// TwinCAT 3 PLC project SampleProject
// ProgramVersion: 3.1.4022.1
// libraries:
//   Tc2_Standard, * (Beckhoff Automation GmbH)
//   Tc2_System, * (Beckhoff Automation GmbH)
//   Tc2_Utilities, * (Beckhoff Automation GmbH)
//   Tc3_Module, * (Beckhoff Automation GmbH)
//   Tc3_PLCopen_OpcUa, * (Beckhoff Automation GmbH)
// project tree:
//   / PlcTask.TcTTO
//   POUs/ MAIN.TcPOU, PRG_HA_SingleNode.TcPOU
//   POUs/Multiple Nodes/ FB_HistoryUpdate_INT.TcPOU, FB_HistoryUpdate_LREAL.TcPOU, PRG_HA_MultipleNodes.TcPOU
// real-time tasks:
//   TASK PlcTask: cycle T#10ms, priority 20, ADS port 350

CONFIGURATION SampleProject
    RESOURCE PLC ON TwinCAT3
        TASK PlcTask(INTERVAL := T#10ms, PRIORITY := 20);
        PROGRAM MAIN WITH PlcTask : MAIN;
    END_RESOURCE
END_CONFIGURATION

// ---- POUs/MAIN.TcPOU
PROGRAM MAIN
VAR
	i : INT;
END_VAR

i := i + 1;

PRG_HA_SingleNode();	// call sample for UA_HistoryUpdate
PRG_HA_MultipleNodes();	// call sample for UA_HistoryUpdate with multiple nodes

END_PROGRAM

// ---- POUs/PRG_HA_SingleNode.TcPOU
//| use case:
//| One variable is specified for historical access. 
//| Its values of each task cycle should be updated to data storage.
PROGRAM PRG_HA_SingleNode
VAR CONSTANT
	// These connection and namespace settings need to be adapted to the runtime environment
	cOpcUaServerUrl		: STRING(MAX_STRING_LENGTH) := 'opc.tcp://localhost:4840';
	cNamespaceUri		: STRING(MAX_STRING_LENGTH) := 'urn:BeckhoffAutomation:Ua:PLC1';
	cBufferSize			: UINT := 1000;
END_VAR
VAR
	// Variable for HistorcalAccess
	{attribute 'OPC.UA.DA' := '1'}
	nMyValue : INT;	
	
	// state machine declarations 
	nState					: INT;
	bStart					: BOOL;			//Set True to start this sample.
	bSample					: BOOL := TRUE;	//Set True if data should be sampled.
	bStop					: BOOL;			//Set True to stop the sampling and close the connection afterwards.
	bError					: BOOL;
	nErrorID				: DWORD;
	
	// Declarations for UA_Connect
	fbUAConnect				: UA_Connect;
	stSessionConnectInfo 	: ST_UASessionConnectInfo;
	nConnectionHdl			: DWORD;
	
	// Declarations for UA_GetNamespaceIndex
	fbUAGetNamespaceIndex	: UA_GetNamespaceIndex;
	nNamespaceIndex			: UINT;
	
	// Declarations for UA_NodeGetHandle
	fbUANodeGetHandle		: UA_NodeGetHandle;
	sNodeIdentifier			: STRING(MAX_STRING_LENGTH) := 'PRG_HA_SingleNode.nMyValue'; // change to node identifier
	NodeID					: ST_UANodeID;
	nNodeHdl				: DWORD;
	
	// Declarations for UA_HistoryUpdate
	fbUAHistoryUpdate		: UA_HistoryUpdate;
	aDataValues				: ARRAY [1..cBufferSize] OF UAHADataValue(ValueSize:=SIZEOF(nMyValue));
	aValueErrorIDs			: ARRAY [1..cBufferSize] OF DWORD;
	nCounter				: UINT := 1;
	
	// Declarations for UA_NodeReleaseHandle
	fbUANodeReleaseHandle	: UA_NodeReleaseHandle;
	
	// Declarations for UA_Disconnect
	fbUADisconnect			: UA_Disconnect;
END_VAR

nMyValue := nMyValue + 1;

CASE nState OF
0:	//Idle
	IF bStart THEN  // the opc ua server need to be startet
		bStart				:= FALSE;
		bError				:= FALSE;
		nErrorID			:= 0;
		nCounter			:= 1;

		stSessionConnectInfo.tConnectTimeout 		:= T#1M;
		stSessionConnectInfo.tSessionTimeout 		:= T#1M;
		stSessionConnectInfo.sApplicationName		:= '';
		stSessionConnectInfo.eSecurityMode 			:= eUASecurityMsgMode_None;
		stSessionConnectInfo.eSecurityPolicyUri 	:= eUASecurityPolicy_None;
		stSessionConnectInfo.eTransportProfileUri	:= eUATransportProfileUri_UATcp;
		
		nState := 1;
	END_IF

1: //Open UA Session
	fbUAConnect(	Execute 			:= TRUE,
					ServerUrl			:= cOpcUaServerUrl,
					SessionConnectInfo	:= stSessionConnectInfo,
					Timeout				:= T#5S,
					ConnectionHdl 		=> nConnectionHdl );
		
	IF NOT fbUAConnect.Busy THEN
		IF NOT fbUAConnect.Error THEN
			nState 			:= 2;
		ELSE
			bError 			:= TRUE;
			nErrorID		:= fbUAConnect.ErrorID;
			nConnectionHdl 	:= 0;
			nState 			:= 0; //Idle
		END_IF
		fbUAConnect(Execute := FALSE);
	END_IF

2: //Get NS Index
	fbUAGetNamespaceIndex(	Execute 			:= TRUE,
							ConnectionHdl		:= nConnectionHdl,
							NamespaceUri		:= cNamespaceUri,
							NamespaceIndex		=> nNamespaceIndex );
		
	IF NOT fbUAGetNamespaceIndex.Busy THEN
		IF NOT fbUAGetNamespaceIndex.Error THEN
			nState 			:= 3;
		ELSE
			bError 			:= TRUE;
			nErrorID		:= fbUAGetNamespaceIndex.ErrorID;
			nState			:= 6; //Close Connection
		END_IF
		fbUAGetNamespaceIndex(Execute := FALSE);
	END_IF
	
3: //Get Node Handle
	NodeID.eIdentifierType 	:= eUAIdentifierType_String;
	NodeID.nNamespaceIndex 	:= nNamespaceIndex;
	NodeID.sIdentifier		:= sNodeIdentifier;
	
	fbUANodeGetHandle(	Execute 			:= TRUE,
						ConnectionHdl 		:= nConnectionHdl,
						NodeID 				:= NodeID,
						NodeHdl				=> nNodeHdl );
		
	IF NOT fbUANodeGetHandle.Busy THEN
		IF NOT fbUANodeGetHandle.Error THEN
			nState 			:= 4;
		ELSE
			bError  		:= TRUE;
			nErrorID 		:= fbUANodeGetHandle.ErrorID;
			nState 			:= 6; //Close Connection
		END_IF
		fbUANodeGetHandle(Execute := FALSE);
	END_IF
	
4: //UA_HistoryUpdate
	IF bSample THEN
		aDataValues[nCounter].Value				:= ADR(nMyValue);
		aDataValues[nCounter].StatusCode 		:= UAHAUpdateStatusCode.HistorianRaw;
		aDataValues[nCounter].ServerTimeStamp 	:= F_GetSystemTime();
		aDataValues[nCounter].SourceTimeStamp 	:= aDataValues[nCounter].ServerTimeStamp;	
		nCounter := nCounter + 1;
		
		IF nCounter > cBufferSize THEN
			fbUAHistoryUpdate.Execute := TRUE;
			nCounter := 1;
		END_IF
	END_IF
	
	fbUAHistoryUpdate(	Execute 			:= , //already set above
						ConnectionHdl 		:= nConnectionHdl,
						NodeHdl 			:= nNodeHdl,
						PerformInsert 		:= TRUE,
						PerformReplace 		:= FALSE,
						DataValueCount 		:= cBufferSize,
						DataValues	 		:= aDataValues,
						ValueErrorIDs 		:= aValueErrorIDs );
						
	IF NOT fbUAHistoryUpdate.Busy THEN
		IF NOT fbUAHistoryUpdate.Error THEN 
			IF bStop THEN
				bStop		:= FALSE;
				nState 		:= 5;
			END_IF
		ELSE
			bError 			:= TRUE;
			nErrorID 		:= fbUAHistoryUpdate.ErrorID;
			nState 			:= 5; //Release Node Handle
		END_IF
		fbUAHistoryUpdate(	Execute			:= FALSE, 			
							DataValues	 	:= aDataValues,
							ValueErrorIDs 	:= aValueErrorIDs);
	END_IF

5: //Release Node Handle
	fbUANodeReleaseHandle(	Execute 			:= TRUE,
							ConnectionHdl 		:= nConnectionHdl,
							NodeHdl 			:= nNodeHdl );
		
	IF NOT fbUANodeReleaseHandle.Busy THEN
		IF fbUANodeReleaseHandle.Error THEN
			bError 		:= TRUE;
			nErrorID 	:= fbUANodeReleaseHandle.ErrorID;
		END_IF
		fbUANodeReleaseHandle(Execute := FALSE);
		nState 			:= 6; //Close Connection
	END_IF

6: //Close Session
	fbUADisconnect( Execute := TRUE, ConnectionHdl := nConnectionHdl );
		
	IF NOT fbUADisconnect.Busy THEN
		IF fbUADisconnect.Error THEN
			bError 			:= TRUE;
			nErrorID 		:= fbUADisconnect.ErrorID;
			nConnectionHdl 	:= 0;
		END_IF
		fbUADisconnect(Execute := FALSE);
		nState := 0;
	END_IF
END_CASE

END_PROGRAM

// ---- POUs/Multiple Nodes/PRG_HA_MultipleNodes.TcPOU
//| use case:
//| Three variables are specified for historical access. 
//| Every three seconds their values should be updated to data storage for one second long.
PROGRAM PRG_HA_MultipleNodes
VAR CONSTANT
	// These connection and namespace settings need to be adapted to the runtime environment
	cOpcUaServerUrl			: STRING(MAX_STRING_LENGTH) := 'opc.tcp://localhost:4840';
	cNamespaceUri			: STRING(MAX_STRING_LENGTH) := 'urn:BeckhoffAutomation:Ua:PLC1';
END_VAR
VAR
	// Variables for HistorcalAccess
	{attribute 'OPC.UA.DA' := '1'}
	nMyValue1 : INT;	
	{attribute 'OPC.UA.DA' := '1'}
	nMyValue2 : INT;
	{attribute 'OPC.UA.DA' := '1'}
	fMyValue3 : LREAL;
	
	// state machine declarations 
	nState					: INT;
	bStart					: BOOL;  		//Set True to start this sample.
	bSample					: BOOL;			//Set True to stop the sampling.
	bStop					: BOOL;			//Set True to close the connection afterwards.
	bError					: BOOL;
	nErrorID				: DWORD;
	fbTimer					: TON:=(PT:=T#3S);
	
	// Declarations for UA_Connect
	fbUAConnect				: UA_Connect;
	stSessionConnectInfo 	: ST_UASessionConnectInfo;
	nConnectionHdl			: DWORD;
	
	// Declarations for UA_GetNamespaceIndex
	fbUAGetNamespaceIndex	: UA_GetNamespaceIndex;
	nNamespaceIndex			: UINT;
	
	// Declarations for UA_HistoryUpdate
	fbHistoryUpdateNode1	: FB_HistoryUpdate_INT := (sNodeIdentifier := 'PRG_HA_MultipleNodes.nMyValue1');
	fbHistoryUpdateNode2	: FB_HistoryUpdate_INT := (sNodeIdentifier := 'PRG_HA_MultipleNodes.nMyValue2');
	fbHistoryUpdateNode3	: FB_HistoryUpdate_LREAL := (sNodeIdentifier := 'PRG_HA_MultipleNodes.fMyValue3');
	
	// Declarations for UA_Disconnect
	fbUADisconnect			: UA_Disconnect;
	
END_VAR

nMyValue1 := nMyValue1 + 1;
nMyValue2 := nMyValue2 + 2;
fMyValue3 := fMyValue3 + 1.5;

CASE nState OF
0:	//Idle
	IF bStart THEN
		bStart				:= FALSE;
		bError				:= FALSE;
		nErrorID			:= 0;

		stSessionConnectInfo.tConnectTimeout 		:= T#1M;
		stSessionConnectInfo.tSessionTimeout 		:= T#1M;
		stSessionConnectInfo.sApplicationName		:= '';
		stSessionConnectInfo.eSecurityMode 			:= eUASecurityMsgMode_None;
		stSessionConnectInfo.eSecurityPolicyUri 	:= eUASecurityPolicy_None;
		stSessionConnectInfo.eTransportProfileUri	:= eUATransportProfileUri_UATcp;
		
		nState := 1;
	END_IF

1: //Open UA Session
	fbUAConnect(	Execute 			:= TRUE,
					ServerUrl			:= cOpcUaServerUrl,
					SessionConnectInfo	:= stSessionConnectInfo,
					Timeout				:= T#5S,
					ConnectionHdl 		=> nConnectionHdl );
		
	IF NOT fbUAConnect.Busy THEN
		IF NOT fbUAConnect.Error THEN
			nState 			:= 2;
		ELSE
			bError 			:= TRUE;
			nErrorID		:= fbUAConnect.ErrorID;
			nConnectionHdl 	:= 0;
			nState 			:= 0; //Idle
		END_IF
		fbUAConnect(Execute := FALSE);
	END_IF

2: //Get NS Index
	fbUAGetNamespaceIndex(	Execute 			:= TRUE,
							ConnectionHdl		:= nConnectionHdl,
							NamespaceUri		:= cNamespaceUri,
							NamespaceIndex		=> nNamespaceIndex );
		
	IF NOT fbUAGetNamespaceIndex.Busy THEN
		IF NOT fbUAGetNamespaceIndex.Error THEN
			nState 			:= 3;
		ELSE
			bError 			:= TRUE;
			nErrorID		:= fbUAGetNamespaceIndex.ErrorID;
			nState			:= 6; //Close Connection
		END_IF
		fbUAGetNamespaceIndex(Execute := FALSE);
	END_IF

3: //Get Node Handle & HistoryUpdate & ReleaseHandle
	//every three seconds the values should be updated for one second long.
	fbTimer(IN:=TRUE);
	IF fbTimer.ET > T#2S THEN
		bSample := TRUE;
	END_IF
	IF fbTimer.Q THEN
		bSample :=FALSE;
		fbTimer(IN:=FALSE);
	END_IF

	fbHistoryUpdateNode1(	bSample:=bSample, bStop:=bStop,	
							nConnectionHdl:=nConnectionHdl, 
							nNamespaceIndex:=nNamespaceIndex, 
							pValue:=ADR(nMyValue1) );
	IF fbHistoryUpdateNode1.bError THEN
		bError 		:= TRUE;
		nErrorID 	:= fbHistoryUpdateNode1.nErrorID;		
	END_IF

	fbHistoryUpdateNode2(	bSample:=bSample, bStop:=bStop,
							nConnectionHdl:=nConnectionHdl, 
							nNamespaceIndex:=nNamespaceIndex, 
							pValue:=ADR(nMyValue2) );
	IF fbHistoryUpdateNode2.bError THEN
		bError 		:= TRUE;
		nErrorID 	:= fbHistoryUpdateNode2.nErrorID;		
	END_IF
	
	fbHistoryUpdateNode3(	bSample:=bSample, bStop:=bStop,
							nConnectionHdl:=nConnectionHdl, 
							nNamespaceIndex:=nNamespaceIndex, 
							pValue:=ADR(fMyValue3) );
	IF fbHistoryUpdateNode2.bError THEN
		bError 		:= TRUE;
		nErrorID 	:= fbHistoryUpdateNode3.nErrorID;		
	END_IF	
	
	IF bStop 	AND NOT fbHistoryUpdateNode1.bBusy AND fbHistoryUpdateNode1.nNodeHdl = 0
				AND NOT fbHistoryUpdateNode2.bBusy AND fbHistoryUpdateNode2.nNodeHdl = 0
				AND NOT fbHistoryUpdateNode3.bBusy AND fbHistoryUpdateNode3.nNodeHdl = 0 THEN
		bStop := FALSE;
		nState := 6; //Close Connection
	END_IF 
	
6: //Close Session
	fbUADisconnect( Execute := TRUE, ConnectionHdl := nConnectionHdl );
		
	IF NOT fbUADisconnect.Busy THEN
		IF fbUADisconnect.Error THEN
			bError 			:= TRUE;
			nErrorID 		:= fbUADisconnect.ErrorID;
			nConnectionHdl 	:= 0;
		END_IF
		fbUADisconnect(Execute := FALSE);
		nState := 0; //Idle
	END_IF
	
END_CASE

END_PROGRAM

// ---- POUs/Multiple Nodes/FB_HistoryUpdate_INT.TcPOU
FUNCTION_BLOCK FB_HistoryUpdate_INT
VAR_INPUT
	bSample			: BOOL := TRUE; //Set True if data should be sampled; set FALSE if sampling should be stopped.
	bStop			: BOOL; // set TRUE if nodes should be released
	nConnectionHdl	: DWORD;
	nNamespaceIndex	: UINT;
	sNodeIdentifier	: STRING(MAX_STRING_LENGTH);
	pValue			: PVOID;
END_VAR
VAR_OUTPUT
	bBusy			: BOOL;
	bError			: BOOL;
	nErrorID		: DWORD;
	nNodeHdl		: DWORD;
END_VAR

VAR CONSTANT
	cBufferSize		: UINT := 1000;
	cValueSize		: UINT := SIZEOF(INT);
END_VAR
VAR
	// state machine declarations 
	RisingEdgeStart			: R_TRIG;
	nState					: INT := 0;

	// Declarations for UA_NodeGetHandle
	fbUANodeGetHandle		: UA_NodeGetHandle;
	NodeID					: ST_UANodeID := (eIdentifierType 	:= eUAIdentifierType_String);
	
	// Declarations for UA_HistoryUpdate
	fbUAHistoryUpdate		: UA_HistoryUpdate;
	aDataValues				: ARRAY [1..cBufferSize] OF UAHADataValue(ValueSize:=cValueSize);
	aValueErrorIDs			: ARRAY [1..cBufferSize] OF DWORD;
	nCounter				: UINT := 1;
	
	// Declarations for UA_NodeReleaseHandle
	fbUANodeReleaseHandle	: UA_NodeReleaseHandle;
END_VAR

RisingEdgeStart(CLK:=bSample);

CASE nState OF
0: //Idle	
	IF RisingEdgeStart.Q THEN
		bError := FALSE;
		nErrorID := 0;
		nCounter := 1;
		
		NodeID.nNamespaceIndex 	:= nNamespaceIndex;
		NodeID.sIdentifier		:= sNodeIdentifier;
		
		fbUANodeGetHandle(	Execute 			:= TRUE,
							ConnectionHdl 		:= nConnectionHdl,
							NodeID 				:= NodeID,
							Busy				=> bBusy );	
		nState := 1;	
	END_IF
	
1: //Get Node Handle
	fbUANodeGetHandle(Execute := FALSE, NodeHdl=>nNodeHdl, Busy=>bBusy );
	IF NOT fbUANodeGetHandle.Busy THEN
		IF NOT fbUANodeGetHandle.Error THEN
			nCounter		:= 1;
			nState 			:= 2;
		ELSE
			bError  		:= TRUE;
			nErrorID 		:= fbUANodeGetHandle.ErrorID;
			nState 			:= 666; //error state
		END_IF
	END_IF
	
2: //UA_HistoryUpdate
	IF bSample THEN
		aDataValues[nCounter].Value			 	:= pValue;
		aDataValues[nCounter].StatusCode 		:= UAHAUpdateStatusCode.HistorianRaw;
		aDataValues[nCounter].ServerTimeStamp 	:= F_GetSystemTime();
		aDataValues[nCounter].SourceTimeStamp 	:= aDataValues[nCounter].ServerTimeStamp;	
		nCounter := nCounter + 1;

		IF nCounter > cBufferSize THEN
			fbUAHistoryUpdate.Execute := TRUE;
			nCounter := 1;
		END_IF
	END_IF
	
	fbUAHistoryUpdate(	Execute 		:= , //already set above
						ConnectionHdl 	:= nConnectionHdl,
						NodeHdl 		:= nNodeHdl,
						PerformInsert 	:= TRUE,
						PerformReplace 	:= FALSE,
						DataValueCount 	:= cBufferSize,
						DataValues	 	:= aDataValues,
						ValueErrorIDs 	:= aValueErrorIDs,
						Busy			=> bBusy );
						
	IF NOT fbUAHistoryUpdate.Busy THEN
		IF NOT fbUAHistoryUpdate.Error THEN
			IF bStop THEN
				nState := 3; //Release Node Handle
			END_IF
		ELSE
			bError 			:= TRUE;
			nErrorID 		:= fbUAHistoryUpdate.ErrorID;
			nState 			:= 666; //error state
		END_IF
		fbUAHistoryUpdate(	Execute			:= FALSE, 			
							DataValues	 	:= aDataValues,
							ValueErrorIDs 	:= aValueErrorIDs,
							Busy			=> bBusy );
	END_IF
	
3: //Release Node Handle
	fbUANodeReleaseHandle(	Execute 		:= TRUE,
							ConnectionHdl 	:= nConnectionHdl,
							NodeHdl 		:= nNodeHdl,
							Busy			=> bBusy );
		
	IF NOT fbUANodeReleaseHandle.Busy THEN
		IF NOT fbUANodeReleaseHandle.Error THEN
			nState		:= 0;
			nNodeHdl	:= 0;
		ELSE
			bError 		:= TRUE;
			nErrorID 	:= fbUANodeReleaseHandle.ErrorID;
			nState 		:= 666; //error state
		END_IF
		fbUANodeReleaseHandle(Execute := FALSE, Busy => bBusy );
	END_IF	
	
666: //error state	
	
END_CASE

END_FUNCTION_BLOCK

// ---- POUs/Multiple Nodes/FB_HistoryUpdate_LREAL.TcPOU
FUNCTION_BLOCK FB_HistoryUpdate_LREAL
VAR_INPUT
	bSample			: BOOL := TRUE; //Set True if data should be sampled; set FALSE if sampling should be stopped.
	bStop			: BOOL; // set TRUE if nodes should be released
	nConnectionHdl	: DWORD;
	nNamespaceIndex	: UINT;
	sNodeIdentifier	: STRING(MAX_STRING_LENGTH);
	pValue			: PVOID;
END_VAR
VAR_OUTPUT
	bBusy			: BOOL;
	bError			: BOOL;
	nErrorID		: DWORD;
	nNodeHdl		: DWORD;
END_VAR

VAR CONSTANT
	cBufferSize		: UINT := 1000;
	cValueSize		: UINT := SIZEOF(LREAL);
END_VAR
VAR
	// state machine declarations 
	RisingEdgeStart			: R_TRIG;
	nState					: INT := 0;

	// Declarations for UA_NodeGetHandle
	fbUANodeGetHandle		: UA_NodeGetHandle;
	NodeID					: ST_UANodeID := (eIdentifierType 	:= eUAIdentifierType_String);
	
	// Declarations for UA_HistoryUpdate
	fbUAHistoryUpdate		: UA_HistoryUpdate;
	aDataValues				: ARRAY [1..cBufferSize] OF UAHADataValue(ValueSize:=cValueSize);
	aValueErrorIDs			: ARRAY [1..cBufferSize] OF DWORD;
	nCounter				: UINT := 1;
	
	// Declarations for UA_NodeReleaseHandle
	fbUANodeReleaseHandle	: UA_NodeReleaseHandle;
END_VAR

RisingEdgeStart(CLK:=bSample);

CASE nState OF
0: //Idle	
	IF RisingEdgeStart.Q THEN
		bError := FALSE;
		nErrorID := 0;
		nCounter := 1;
		
		NodeID.nNamespaceIndex 	:= nNamespaceIndex;
		NodeID.sIdentifier		:= sNodeIdentifier;
		
		fbUANodeGetHandle(	Execute 			:= TRUE,
							ConnectionHdl 		:= nConnectionHdl,
							NodeID 				:= NodeID,
							Busy				=> bBusy );	
		nState := 1;	
	END_IF
	
1: //Get Node Handle
	fbUANodeGetHandle(Execute := FALSE, NodeHdl=>nNodeHdl, Busy=>bBusy );
	IF NOT fbUANodeGetHandle.Busy THEN
		IF NOT fbUANodeGetHandle.Error THEN
			nCounter		:= 1;
			nState 			:= 2;
		ELSE
			bError  		:= TRUE;
			nErrorID 		:= fbUANodeGetHandle.ErrorID;
			nState 			:= 666; //error state
		END_IF
	END_IF
	
2: //UA_HistoryUpdate
	IF bSample THEN
		aDataValues[nCounter].Value			 	:= pValue;
		aDataValues[nCounter].StatusCode 		:= UAHAUpdateStatusCode.HistorianRaw;
		aDataValues[nCounter].ServerTimeStamp 	:= F_GetSystemTime();
		aDataValues[nCounter].SourceTimeStamp 	:= aDataValues[nCounter].ServerTimeStamp;	
		nCounter := nCounter + 1;

		IF nCounter > cBufferSize THEN
			fbUAHistoryUpdate.Execute := TRUE;
			nCounter := 1;
		END_IF
	END_IF
	
	fbUAHistoryUpdate(	Execute 		:= , //already set above
						ConnectionHdl 	:= nConnectionHdl,
						NodeHdl 		:= nNodeHdl,
						PerformInsert 	:= TRUE,
						PerformReplace 	:= FALSE,
						DataValueCount 	:= cBufferSize,
						DataValues	 	:= aDataValues,
						ValueErrorIDs 	:= aValueErrorIDs,
						Busy			=> bBusy );
						
	IF NOT fbUAHistoryUpdate.Busy THEN
		IF NOT fbUAHistoryUpdate.Error THEN
			IF bStop THEN
				nState := 3; //Release Node Handle
			END_IF
		ELSE
			bError 			:= TRUE;
			nErrorID 		:= fbUAHistoryUpdate.ErrorID;
			nState 			:= 666; //error state
		END_IF
		fbUAHistoryUpdate(	Execute			:= FALSE, 			
							DataValues	 	:= aDataValues,
							ValueErrorIDs 	:= aValueErrorIDs,
							Busy			=> bBusy );
	END_IF
	
3: //Release Node Handle
	fbUANodeReleaseHandle(	Execute 		:= TRUE,
							ConnectionHdl 	:= nConnectionHdl,
							NodeHdl 		:= nNodeHdl,
							Busy			=> bBusy );
		
	IF NOT fbUANodeReleaseHandle.Busy THEN
		IF NOT fbUANodeReleaseHandle.Error THEN
			nState		:= 0;
			nNodeHdl	:= 0;
		ELSE
			bError 		:= TRUE;
			nErrorID 	:= fbUANodeReleaseHandle.ErrorID;
			nState 		:= 666; //error state
		END_IF
		fbUANodeReleaseHandle(Execute := FALSE, Busy => bBusy );
	END_IF	
	
666: //error state	
	
END_CASE

END_FUNCTION_BLOCK
